LIN {X 0,Y 119.569,Z 419.202,A -85,B 0,C 180,E1 -30597.748,E2 -30597.748} C_VEL
LIN {X 0,Y 130.053,Z 408.467,A -85,B 0,C 180,E1 -30598.68,E2 -30598.68} C_VEL
LIN {X 0,Y 139.691,Z 396.738,A -85,B 0,C 180,E1 -30599.362,E2 -30599.362} C_VEL
LIN {X 0,Y 140.568,Z 395.569,A -85,B 0,C 180,E1 -30599.428,E2 -30599.428} C_VEL
LIN {X 0,Y 140.565,Z 395.579,A -85,B 0,C 180,E1 -30599.574,E2 -30599.574} C_VEL
LIN {X 0,Y 130.799,Z 407.697,A -85,B 0,C 180,E1 -30600.208,E2 -30600.208} C_VEL
LIN {X 0,Y 121.249,Z 417.758,A -85,B 0,C 180,E1 -30600.896,E2 -30600.896} C_VEL
LIN {X 0,Y 110.743,Z 427.146,A -85,B 0,C 180,E1 -30601.74,E2 -30601.74} C_VEL
LIN {X 0,Y 98.531,Z 436.385,A -85,B 0,C 180,E1 -30603.031,E2 -30603.031} C_VEL
LIN {X 0,Y 84.676,Z 445.095,A -85,B 0,C 180,E1 -30605.131,E2 -30605.131} C_VEL
LIN {X 0,Y 70.973,Z 452.092,A -85,B 0,C 180,E1 -30608.009,E2 -30608.009} C_VEL
LIN {X 0,Y 57.511,Z 457.598,A -85,B 0,C 180,E1 -30612.141,E2 -30612.141} C_VEL
LIN {X 0,Y 44.543,Z 461.773,A -85,B 0,C 180,E1 -30618.794,E2 -30618.794} C_VEL
LIN {X 0,Y 32.573,Z 464.71,A -85,B 0,C 180,E1 -30630.338,E2 -30630.338} C_VEL
LIN {X 0,Y 23.16,Z 466.475,A -85,B 0,C 180,E1 -30652.632,E2 -30652.632} C_VEL
LIN {X 0,Y 19.928,Z 467.098,A -85,B 0,C 180,E1 -30689.999,E2 -30689.999} C_VEL
LIN {X 0,Y 23.144,Z 466.45,A -85,B 0,C 180,E1 -30727.396,E2 -30727.396} C_VEL
LIN {X 0,Y 32.553,Z 464.651,A -85,B 0,C 180,E1 -30749.719,E2 -30749.719} C_VEL
LIN {X 0,Y 45.537,Z 461.388,A -85,B 0,C 180,E1 -30762.022,E2 -30762.022} C_VEL
LIN {X 0,Y 57.498,Z 457.484,A -85,B 0,C 180,E1 -30767.916,E2 -30767.916} C_VEL
LIN {X 0,Y 70.966,Z 451.939,A -85,B 0,C 180,E1 -30772.028,E2 -30772.028} C_VEL
LIN {X 0,Y 84.672,Z 444.896,A -85,B 0,C 180,E1 -30774.898,E2 -30774.898} C_VEL
LIN {X 0,Y 96.789,Z 437.374,A -85,B 0,C 180,E1 -30776.766,E2 -30776.766} C_VEL
LIN {X 0,Y 108.994,Z 428.317,A -85,B 0,C 180,E1 -30778.1,E2 -30778.1} C_VEL
LIN {X 0,Y 119.494,Z 419.076,A -85,B 0,C 180,E1 -30778.999,E2 -30778.999} C_VEL
LIN {X 0,Y 129.686,Z 408.564,A -85,B 0,C 180,E1 -30779.723,E2 -30779.723} C_VEL
LIN {X 0,Y 139.685,Z 396.308,A -85,B 0,C 180,E1 -30780.39,E2 -30780.39} C_VEL
LIN {X 0,Y 140.564,Z 395.132,A -85,B 0,C 180,E1 -30780.437,E2 -30780.437} C_VEL
LIN {X 0,Y 140.569,Z 395.117,A -85,B 0,C 180,E1 -30780.648,E2 -30780.648} C_VEL
LIN {X 0,Y 140.608,Z 397.116,A -85,B 0,C 180,E1 -30781.486,E2 -30781.486} C_VEL
LIN {X 0,Y 140.608,Z 450.399,A -85,B 0,C 180,E1 -30781.486,E2 -30781.486} C_VEL
LIN {X 0,Y 96.406,Z 450.399,A -85,B 0,C 180,E1 -30781.129,E2 -30781.129} C_VEL
LIN {X 0,Y 94.407,Z 448.399,A -85,B 0,C 180,E1 -30781.105,E2 -30781.105} C_VEL
LIN {X 0,Y 94.407,Z 442.215,A -85,B 0,C 180,E1 -30781.105,E2 -30781.105} C_VEL
LIN {X 0,Y 91.39,Z 440.51,A -85,B 0,C 180,E1 -30781.369,E2 -30781.369} C_VEL
LIN {X 0,Y 80.904,Z 446.459,A -85,B 0,C 180,E1 -30782.578,E2 -30782.578} C_VEL
LIN {X 0,Y 67.003,Z 452.997,A -85,B 0,C 180,E1 -30784.823,E2 -30784.823} C_VEL
LIN {X 0,Y 53.257,Z 458.097,A -85,B 0,C 180,E1 -30788.223,E2 -30788.223} C_VEL
LIN {X 0,Y 43.127,Z 461.03,A -85,B 0,C 180,E1 -30792.104,E2 -30792.104} C_VEL
LIN {X 0,Y 30.102,Z 463.889,A -85,B 0,C 180,E1 -30800.953,E2 -30800.953} C_VEL
LIN {X 0,Y 18.648,Z 465.591,A -85,B 0,C 180,E1 -30821.084,E2 -30821.084} C_VEL
LIN {X 0,Y 13.054,Z 466.174,A -85,B 0,C 180,E1 -30870.001,E2 -30870.001} C_VEL
LIN {X 0,Y 18.639,Z 465.618,A -85,B 0,C 180,E1 -30918.951,E2 -30918.951} C_VEL
LIN {X 0,Y 30.072,Z 463.952,A -85,B 0,C 180,E1 -30939.203,E2 -30939.203} C_VEL
LIN {X 0,Y 43.118,Z 461.122,A -85,B 0,C 180,E1 -30947.953,E2 -30947.953} C_VEL
LIN {X 0,Y 56.662,Z 457.065,A -85,B 0,C 180,E1 -30952.874,E2 -30952.874} C_VEL
LIN {X 0,Y 70.462,Z 451.676,A -85,B 0,C 180,E1 -30955.884,E2 -30955.884} C_VEL
LIN {X 0,Y 84.389,Z 444.803,A -85,B 0,C 180,E1 -30957.988,E2 -30957.988} C_VEL
LIN {X 0,Y 91.388,Z 440.737,A -85,B 0,C 180,E1 -30958.706,E2 -30958.706} C_VEL
LIN {X 0,Y 91.368,Z 440.772,A -85,B 0,C 180,E1 -30959.505,E2 -30959.505} C_VEL
LIN {X 0,Y 77.325,Z 448.594,A -85,B 0,C 180,E1 -30961.189,E2 -30961.189} C_VEL
LIN {X 0,Y 63.366,Z 454.819,A -85,B 0,C 180,E1 -30963.425,E2 -30963.425} C_VEL
LIN {X 0,Y 49.565,Z 459.645,A -85,B 0,C 180,E1 -30966.994,E2 -30966.994} C_VEL
LIN {X 0,Y 36.096,Z 463.191,A -85,B 0,C 180,E1 -30973.215,E2 -30973.215} C_VEL
LIN {X 0,Y 23.445,Z 465.534,A -85,B 0,C 180,E1 -30985.934,E2 -30985.934} C_VEL
LIN {X 0,Y 14.022,Z 466.731,A -85,B 0,C 180,E1 -31019.918,E2 -31019.918} C_VEL
LIN {X 0,Y 12.815,Z 466.899,A -85,B 0,C 180,E1 -31049.999,E2 -31049.999} C_VEL
LIN {X 0,Y 17.996,Z 466.25,A -85,B 0,C 180,E1 -31101.356,E2 -31101.356} C_VEL
LIN {X 0,Y 29.596,Z 464.451,A -85,B 0,C 180,E1 -31121.776,E2 -31121.776} C_VEL
LIN {X 0,Y 42.924,Z 461.437,A -85,B 0,C 180,E1 -31130.578,E2 -31130.578} C_VEL
LIN {X 0,Y 56.433,Z 457.282,A -85,B 0,C 180,E1 -31135.067,E2 -31135.067} C_VEL
LIN {X 0,Y 70.331,Z 451.737,A -85,B 0,C 180,E1 -31137.808,E2 -31137.808} C_VEL
LIN {X 0,Y 84.337,Z 444.693,A -85,B 0,C 180,E1 -31139.787,E2 -31139.787} C_VEL
LIN {X 0,Y 91.368,Z 440.547,A -85,B 0,C 180,E1 -31140.548,E2 -31140.548} C_VEL
LIN {X 0,Y 91.39,Z 440.51,A -85,B 0,C 180,E1 -31141.369,E2 -31141.369} C_VEL
LIN {X 0,Y 91.462,Z 442.509,A -85,B 0,C 180,E1 -31142.657,E2 -31142.657} C_VEL
LIN {X 0,Y 91.462,Z 469.424,A -85,B 0,C 180,E1 -31142.657,E2 -31142.657} C_VEL
LIN {X 0,Y 52.466,Z 469.424,A -85,B 0,C 180,E1 -31140.88,E2 -31140.88} C_VEL
LIN {X 0,Y 50.471,Z 467.424,A -85,B 0,C 180,E1 -31140.716,E2 -31140.716} C_VEL
LIN {X 0,Y 50.471,Z 461.646,A -85,B 0,C 180,E1 -31140.716,E2 -31140.716} C_VEL
LIN {X 0,Y 48.008,Z 459.709,A -85,B 0,C 180,E1 -31141.209,E2 -31141.209} C_VEL
LIN {X 0,Y 35.248,Z 462.809,A -85,B 0,C 180,E1 -31144.482,E2 -31144.482} C_VEL
LIN {X 0,Y 21.546,Z 465.081,A -85,B 0,C 180,E1 -31151.888,E2 -31151.888} C_VEL
LIN {X 0,Y 9.028,Z 466.224,A -85,B 0,C 180,E1 -31178.879,E2 -31178.879} C_VEL
LIN {X 0,Y 5.959,Z 466.373,A -85,B 0,C 180,E1 -31230.003,E2 -31230.003} C_VEL
LIN {X 0,Y 14.957,Z 465.817,A -85,B 0,C 180,E1 -31300.01,E2 -31300.01} C_VEL
LIN {X 0,Y 28.334,Z 464.151,A -85,B 0,C 180,E1 -31312.833,E2 -31312.833} C_VEL
LIN {X 0,Y 42.21,Z 461.321,A -85,B 0,C 180,E1 -31317.454,E2 -31317.454} C_VEL
LIN {X 0,Y 48.025,Z 459.808,A -85,B 0,C 180,E1 -31318.881,E2 -31318.881} C_VEL
LIN {X 0,Y 35.157,Z 462.992,A -85,B 0,C 180,E1 -31321.783,E2 -31321.783} C_VEL
LIN {X 0,Y 21.31,Z 465.334,A -85,B 0,C 180,E1 -31328.35,E2 -31328.35} C_VEL
LIN {X 0,Y 8.625,Z 466.531,A -85,B 0,C 180,E1 -31355.429,E2 -31355.429} C_VEL
LIN {X 0,Y 5.693,Z 466.699,A -85,B 0,C 180,E1 -31409.997,E2 -31409.997} C_VEL
LIN {X 0,Y 14.635,Z 466.049,A -85,B 0,C 180,E1 -31483.826,E2 -31483.826} C_VEL
LIN {X 0,Y 28.189,Z 464.249,A -85,B 0,C 180,E1 -31495.759,E2 -31495.759} C_VEL
LIN {X 0,Y 42.168,Z 461.281,A -85,B 0,C 180,E1 -31500.149,E2 -31500.149} C_VEL
LIN {X 0,Y 48.008,Z 459.709,A -85,B 0,C 180,E1 -31501.209,E2 -31501.209} C_VEL
LIN {X 0,Y 50.502,Z 461.642,A -85,B 0,C 180,E1 -31501.587,E2 -31501.587} C_VEL
LIN {X 0,Y 50.502,Z 600,A -85,B 0,C 180,E1 -31501.587,E2 -31501.587} C_VEL
LIN {X 0,Y 50.502,Z 600,A -85,B 0,C 180,E1 -31501.587,E2 -31501.587}

QRS_NEXT_CUT()

QRS_NEXT()
QRS_HOME()

END
